(* Logix 5000 project; controller ARS14002_PLC vendor 1 type 14 code 218 rev 30.11; software revision 30.01; part 9 of 13 *)
(* tags used below, declared in another part *)
   AN_1000A : CM_AI_SCL;
   AN_1000A_RESTART_TMR : TIMER;
   AN_1000A_SP : REAL;
   AN_1000A_SPL : REAL;
   AN_1000A_STOP_TMR : TIMER;
   AN_1000B : CM_AI_SCL;
   AN_1000B_RESTART_TMR : TIMER;
   AN_1000B_SP : REAL;
   AN_1000B_SPL : REAL;
   AN_1000B_STOP_TMR : TIMER;
   ARS_DERIME_AUTO : BOOL;
   ARS_DERIME_AUTO_OSF_OB : BOOL;
   ARS_DERIME_AUTO_OSF_SB : BOOL;
   ARS_RETURN_AUTO : BOOL;
   AT2_ATOMIZE_FLOW_SCFM : REAL;
   AT2_INLET_FLOW_SCFM : REAL;
   AT2_NONATOMIZE_FLOW : REAL;
   AT2_PLANT_ATOMIZING : BOOL;
   AT2_PLANT_RETURN_AUTO : BOOL;
   AT3_ATOMIZE_FLOW_SCFM : REAL;
   AT3_INLET_FLOW_SCFM : REAL;
   AT3_NONATOMIZE_FLOW : REAL;
   AT3_PLANT_ATOMIZING : BOOL;
   AT3_PLANT_RETURN_AUTO : BOOL;
   BLENDING_OVERRIDE : BOOL;
   CALC_AN_1000B_BLENDED : REAL;
   CALC_HMI_FLOW : REAL;
   CP_Hi_Press_Shutoff : BOOL;
   DEOXO_ARGON_PURGE_DEPRESS : BOOL;
   DEOXO_ARGON_PURGE_FILL : BOOL;
   DEOXO_ARGON_PURGE_HIFLOW : BOOL;
   DEOXO_ARGON_PURGE_LOFLOW : BOOL;
   Deoxo_CurrentState : DINT;
   DEOXO_DEPRESS_TON : TIMER;
   DEOXO_DRY_REM : DINT;
   DEOXO_DRY_TON : TIMER;
   DEOXO_EXOTHERM_SP : REAL;
   DEOXO_OVERTEMP : BOOL;
   DEOXO_OVERTEMP_SPH : REAL;
   DEOXO_OVERTEMP_SPL : REAL;
   DEOXO_POST_EXO_REM : DINT;
   DEOXO_POST_EXOTHERM_TON : TIMER;
   DEOXO_PREHEAT_SP : REAL;
   DEOXO_PURGE_CYC_REM : DINT;
   DEOXO_PURGE_CYCLE_CTU : COUNTER;
   DEOXO_REGEN_HMI_BIT : BOOL;
   DEOXO_REGEN_HMI_BIT_ONS_F : BOOL;
   DEOXO_REGEN_HMI_BIT_ONS_R : BOOL;
   DEOXO_REGEN_RESET : BOOL;
   DEOXO_REGEN_RESET_ONS : BOOL;
   DEOXO_REGEN_RUN : BOOL;
   DEOXO_REGEN_START_PB : BOOL;
   DEOXO_REGEN_STOP_PB : BOOL;
   Deoxo_TransitionState : DINT;
   DEOXO_VENT_SPL : REAL;
   DEOXO_VENT_SWITCH_SP : REAL;
   EN_1250 : BOOL;   // HXR-1250 Enable Signal
   ESTOP_TRIP : BOOL;
   FCV_1001_ENABLE_TON : TIMER;
   FCV_1001_STARTPOS : REAL;
   FCV_1002_Atomize_Mode : BOOL;
   FCV_1002_FLOW_MODE : BOOL;   // 1 = FLOW CONTROL FT-1002 0 = PRESSURE CONTROL PT-1003
   FCV_1002_FLOW_MODE_AN_100B_PPM_MAX : REAL;
   FCV_1002_FLOW_MODE_MIN_FLOW : REAL;
   FCV_1002_FLOW_MODE_N2_PPM_SP : REAL;
   FCV_1002_FLOW_NOT_ATOMIZE_SP : REAL;
   FCV_1002_FLOW_SP : REAL;
   FCV_1002_FLOW_SP_AUTO : BOOL;
   FCV_1002_HIGHPRESS_MAXOPEN : REAL;
   FCV_1002_PT_1003_HIGHALM : BOOL;
   FCV_1002_PT_1003_HIGHLIM : REAL;
   FCV_1002_PT_1003_HIGHLIM_RESET : REAL;
   FCV_1002_PVSWITCH_AUTO : BOOL;
   FCV_1002_SP_Atomize : REAL;
   FCV_1002_SP_Idle_Standby : REAL;
   FCV_1002_STARTPOS : REAL;
   FT_1002 : CM_AI_SCL;
   FT_1002_MAVE : REAL;
   FT_202_ALT_SCFM : REAL;
   HXR_1250 : CM_DO_FVNR;
   LP_SHUTOFF_SPL : REAL;
   MODE_ATOMIZE : BOOL;
   P_800A_Start_Vent_TMR : TIMER;
   P_800B_Start_Vent_TMR : TIMER;
   PIDE_1001 : PID_ENHANCED;
   PIDE_1002 : PID_ENHANCED;
   PIDE_1002_FLOW_IGAIN : REAL;
   PIDE_1002_FLOW_PGAIN : REAL;
   PIDE_1002_FLOW_SP : PID_ENHANCED;
   PIDE_1002_PRESSURE_IGAIN : REAL;
   PIDE_1002_PRESSURE_PGAIN : REAL;
   PIDE_1002_PVCHANGE0 : BOOL;
   PIDE_1002_PVCHANGE1 : BOOL;
   PIDE_1002_RESET : BOOL;
   PIDE_1221 : PID_ENHANCED;
   PIDE_1251 : PID_ENHANCED;
   PIDE_800 : PID_ENHANCED;
   PIDE_800_InRange : BOOL;
   PILOT_PLANT_ATOMIZING : BOOL;
   PILOT_PLANT_RETURN_AUTO : BOOL;
   PRAX_N2_ASSUME : REAL;
   PT_1001 : CM_AI_SCL;
   PT_1001_MINUS_10 : REAL;
   PT_1001_MINUS_50 : REAL;
   PT_1003 : CM_AI_SCL;
   PT_1201 : CM_AI_SCL;
   PT_1301A : CM_AI_SCL;
   PT_902 : CM_AI_SCL;
   PWHMI_StartAtomizing : TIMER;
   Return_Stop_N2 : BOOL;
   Return_Stop_O2 : BOOL;
   SV_1001F : CM_DO_GENERIC;
   SV_1002F : CM_DO_GENERIC;
   SV_1207X : CM_DO_GENERIC;
   SV_1208X : CM_DO_GENERIC;
   SV_1221F : CM_DO_GENERIC;
   SV_1251F : CM_DO_GENERIC;
   TE_1201 : CM_AI_SCL;
   TE_1202 : CM_AI_SCL;
   TE_1203 : CM_AI_SCL;
   TE_901 : CM_AI_SCL;
   TE_901_InRange : BOOL;
   TE_901_SPH : REAL;
   TE_901_SPL : REAL;
   TE_902 : CM_AI_SCL;
   VFD_800A_EN : BOOL;
   VFD_800B_EN : BOOL;
   XV_1001 : CM_DO_VLV;
   XV_1201 : CM_DO_VLV;
   XV_1202 : CM_DO_VLV;
   XV_1203 : CM_DO_VLV;
   XV_1204 : CM_DO_VLV;
   XV_1205 : CM_DO_VLV;
(* MainProgram, continued *)

ROUTINE _306_HP_Product   (* ladder *)
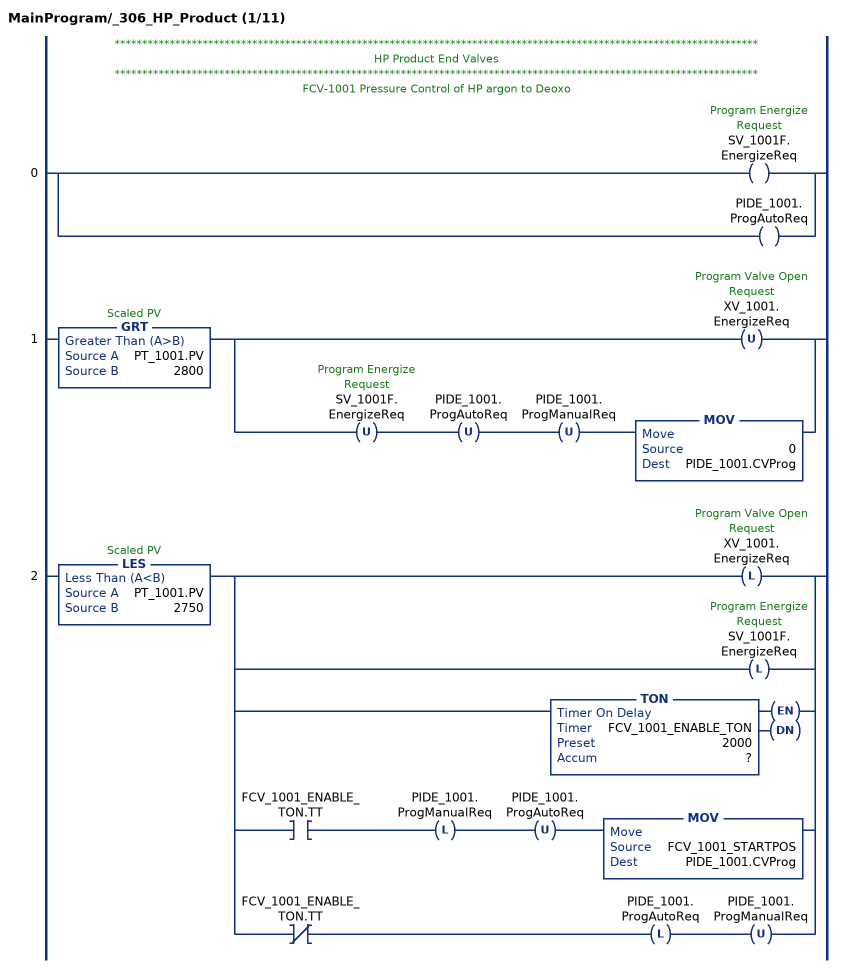
   // *********************************************************************************************************************
   // HP Product End Valves
   // *********************************************************************************************************************
   // FCV-1001 Pressure Control of HP argon to Deoxo
   0: [OTE(SV_1001F.EnergizeReq) ,OTE(PIDE_1001.ProgAutoReq) ];
   1: GRT(PT_1001.PV,2800)[OTU(XV_1001.EnergizeReq) ,OTU(SV_1001F.EnergizeReq) OTU(PIDE_1001.ProgAutoReq) OTU(PIDE_1001.ProgManualReq) MOV(0,PIDE_1001.CVProg) ];
   2: LES(PT_1001.PV,2750)[OTL(XV_1001.EnergizeReq) ,OTL(SV_1001F.EnergizeReq) ,TON(FCV_1001_ENABLE_TON,?,?) ,XIC(FCV_1001_ENABLE_TON.TT) OTL(PIDE_1001.ProgManualReq) OTU(PIDE_1001.ProgAutoReq) MOV(FCV_1001_STARTPOS,PIDE_1001.CVProg) ,XIO(FCV_1001_ENABLE_TON.TT) OTL(PIDE_1001.ProgAutoReq) OTU(PIDE_1001.ProgManualReq) ];
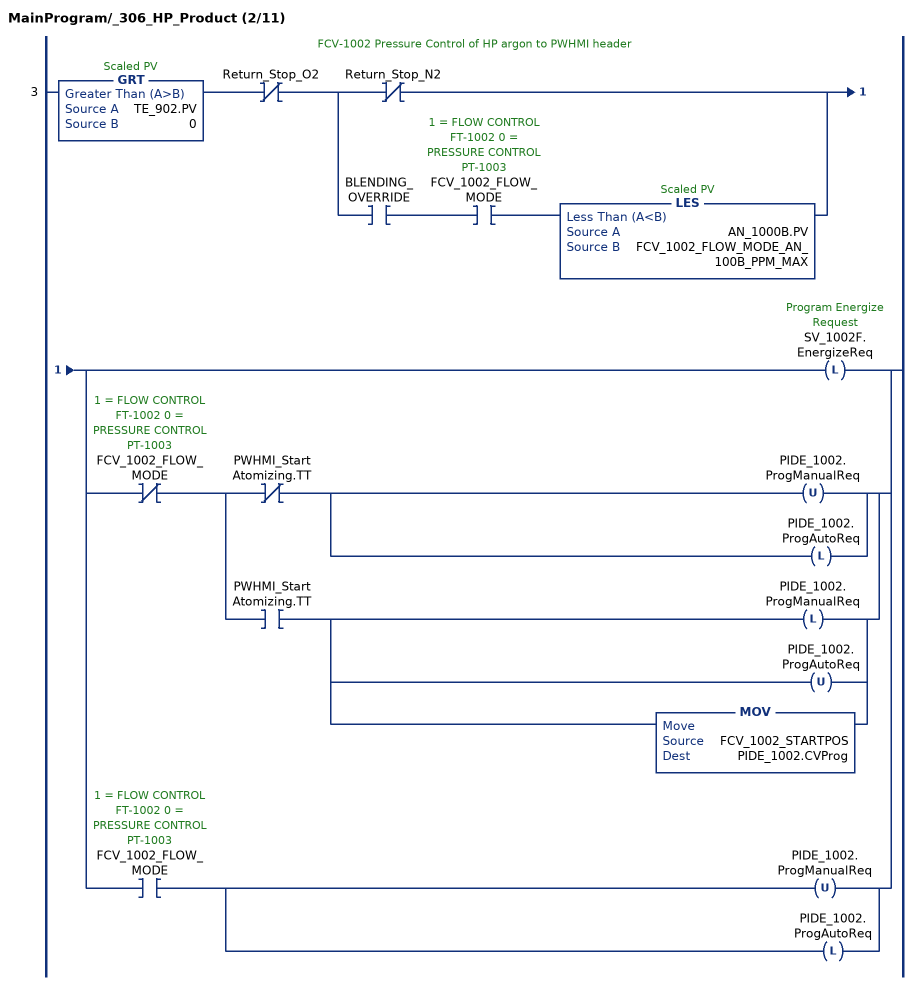
   // FCV-1002 Pressure Control of HP argon to PWHMI header
   3: GRT(TE_902.PV,0)XIO(Return_Stop_O2)[XIO(Return_Stop_N2) ,XIC(BLENDING_OVERRIDE) XIC(FCV_1002_FLOW_MODE) LES(AN_1000B.PV,FCV_1002_FLOW_MODE_AN_100B_PPM_MAX) ][OTL(SV_1002F.EnergizeReq) ,XIO(FCV_1002_FLOW_MODE) [XIO(PWHMI_StartAtomizing.TT) [OTU(PIDE_1002.ProgManualReq) ,OTL(PIDE_1002.ProgAutoReq) ] ,XIC(PWHMI_StartAtomizing.TT) [OTL(PIDE_1002.ProgManualReq) ,OTU(PIDE_1002.ProgAutoReq) ,MOV(FCV_1002_STARTPOS,PIDE_1002.CVProg) ] ] ,XIC(FCV_1002_FLOW_MODE) [OTU(PIDE_1002.ProgManualReq) ,OTL(PIDE_1002.ProgAutoReq) ] ];
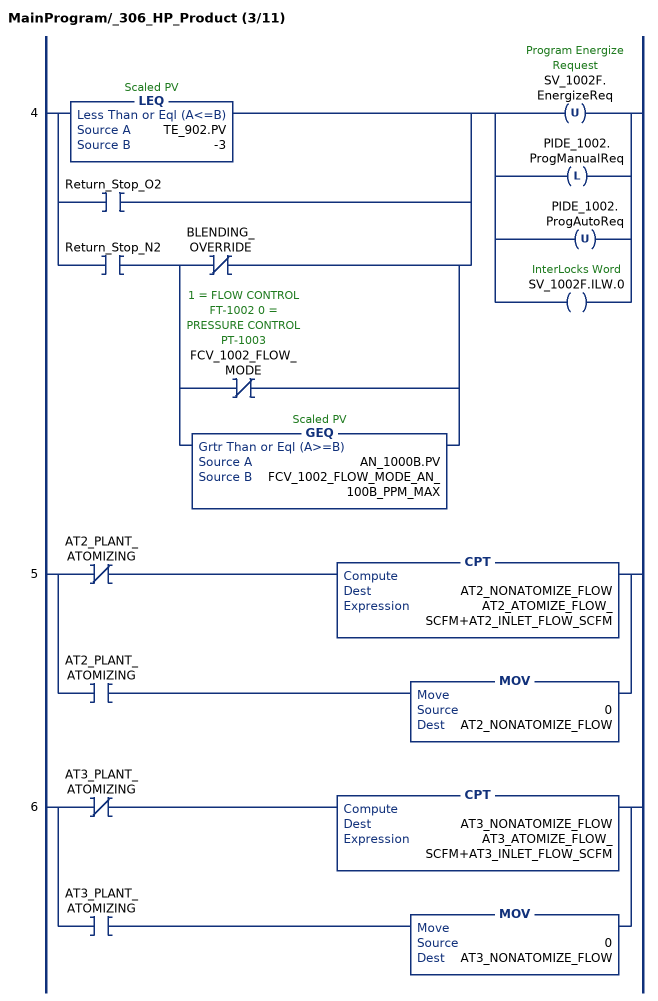
   4: [LEQ(TE_902.PV,-3) ,XIC(Return_Stop_O2) ,XIC(Return_Stop_N2) [XIO(BLENDING_OVERRIDE) ,XIO(FCV_1002_FLOW_MODE) ,GEQ(AN_1000B.PV,FCV_1002_FLOW_MODE_AN_100B_PPM_MAX) ] ][OTU(SV_1002F.EnergizeReq) ,OTL(PIDE_1002.ProgManualReq) ,OTU(PIDE_1002.ProgAutoReq) ,OTE(SV_1002F.ILW.0) ];
   5: [XIO(AT2_PLANT_ATOMIZING) CPT(AT2_NONATOMIZE_FLOW,AT2_ATOMIZE_FLOW_SCFM+AT2_INLET_FLOW_SCFM) ,XIC(AT2_PLANT_ATOMIZING) MOV(0,AT2_NONATOMIZE_FLOW) ];
   6: [XIO(AT3_PLANT_ATOMIZING) CPT(AT3_NONATOMIZE_FLOW,AT3_ATOMIZE_FLOW_SCFM+AT3_INLET_FLOW_SCFM) ,XIC(AT3_PLANT_ATOMIZING) MOV(0,AT3_NONATOMIZE_FLOW) ];
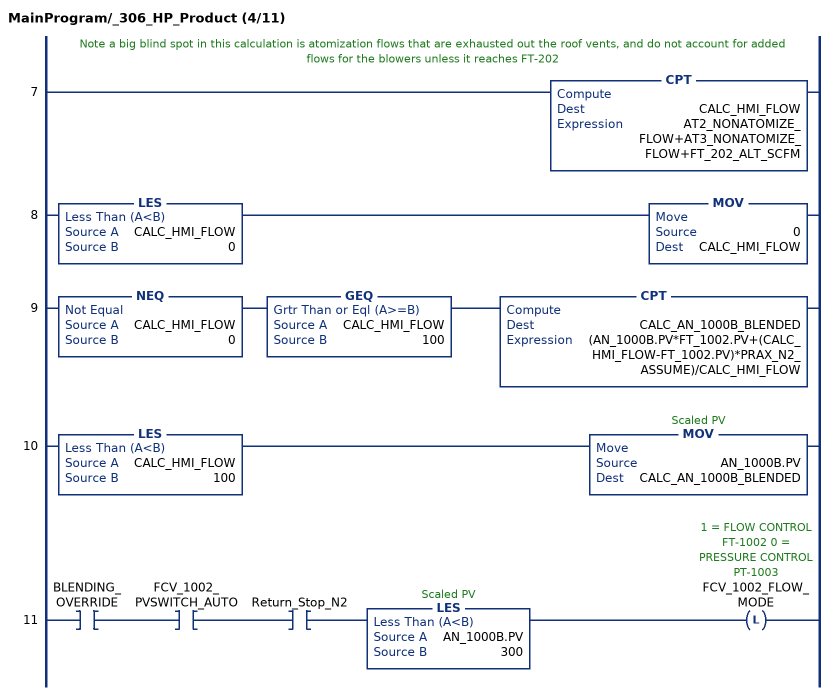
   // Note a big blind spot in this calculation is atomization flows that are exhausted out the roof vents, and do not account for added flows for the blowers unless it reaches FT-202
   7: CPT(CALC_HMI_FLOW,AT2_NONATOMIZE_FLOW+AT3_NONATOMIZE_FLOW+FT_202_ALT_SCFM);
   8: LES(CALC_HMI_FLOW,0)MOV(0,CALC_HMI_FLOW);
   9: NEQ(CALC_HMI_FLOW,0)GEQ(CALC_HMI_FLOW,100)CPT(CALC_AN_1000B_BLENDED,(AN_1000B.PV*FT_1002.PV+(CALC_HMI_FLOW-FT_1002.PV)*PRAX_N2_ASSUME)/CALC_HMI_FLOW);
   10: LES(CALC_HMI_FLOW,100)MOV(AN_1000B.PV,CALC_AN_1000B_BLENDED);
   11: XIC(BLENDING_OVERRIDE)XIC(FCV_1002_PVSWITCH_AUTO)XIC(Return_Stop_N2)LES(AN_1000B.PV,300)OTL(FCV_1002_FLOW_MODE);
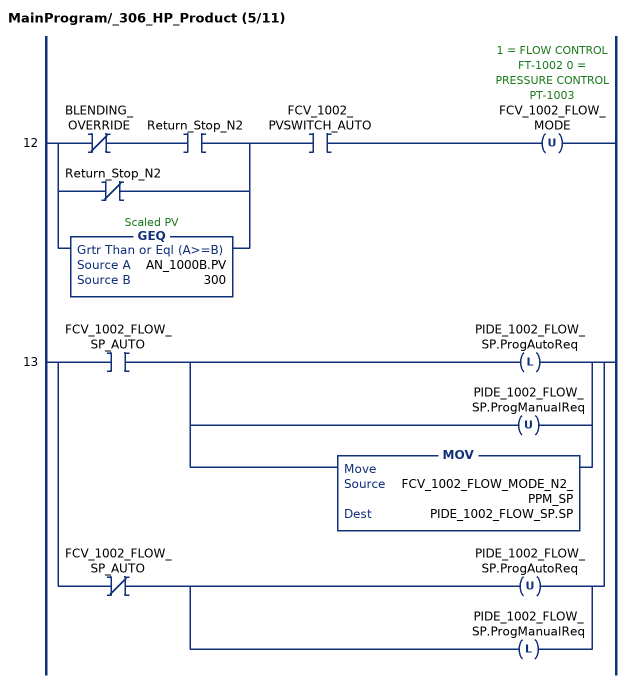
   12: [XIO(BLENDING_OVERRIDE) XIC(Return_Stop_N2) ,XIO(Return_Stop_N2) ,GEQ(AN_1000B.PV,300) ]XIC(FCV_1002_PVSWITCH_AUTO)OTU(FCV_1002_FLOW_MODE);
   13: [XIC(FCV_1002_FLOW_SP_AUTO) [OTL(PIDE_1002_FLOW_SP.ProgAutoReq) ,OTU(PIDE_1002_FLOW_SP.ProgManualReq) ,MOV(FCV_1002_FLOW_MODE_N2_PPM_SP,PIDE_1002_FLOW_SP.SP) ] ,XIO(FCV_1002_FLOW_SP_AUTO) [OTU(PIDE_1002_FLOW_SP.ProgAutoReq) ,OTL(PIDE_1002_FLOW_SP.ProgManualReq) ] ];
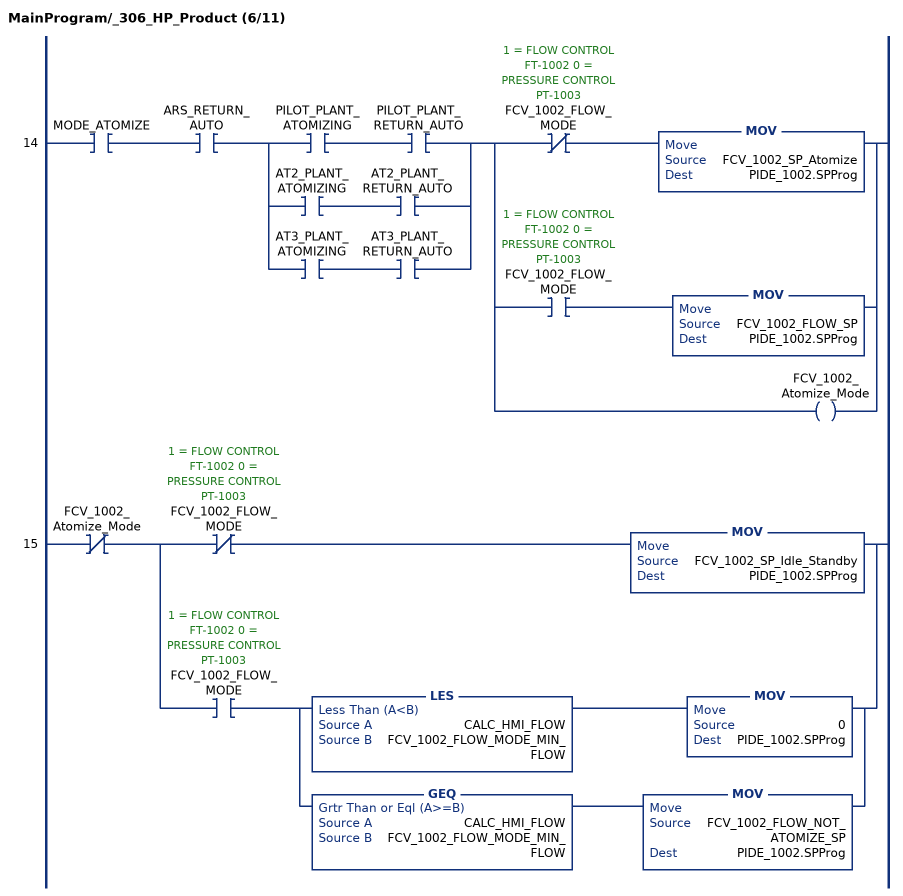
   14: XIC(MODE_ATOMIZE)XIC(ARS_RETURN_AUTO)[XIC(PILOT_PLANT_ATOMIZING) XIC(PILOT_PLANT_RETURN_AUTO) ,XIC(AT2_PLANT_ATOMIZING) XIC(AT2_PLANT_RETURN_AUTO) ,XIC(AT3_PLANT_ATOMIZING) XIC(AT3_PLANT_RETURN_AUTO) ][XIO(FCV_1002_FLOW_MODE) MOV(FCV_1002_SP_Atomize,PIDE_1002.SPProg) ,XIC(FCV_1002_FLOW_MODE) MOV(FCV_1002_FLOW_SP,PIDE_1002.SPProg) ,OTE(FCV_1002_Atomize_Mode) ];
   15: XIO(FCV_1002_Atomize_Mode)[XIO(FCV_1002_FLOW_MODE) MOV(FCV_1002_SP_Idle_Standby,PIDE_1002.SPProg) ,XIC(FCV_1002_FLOW_MODE) [LES(CALC_HMI_FLOW,FCV_1002_FLOW_MODE_MIN_FLOW) MOV(0,PIDE_1002.SPProg) ,GEQ(CALC_HMI_FLOW,FCV_1002_FLOW_MODE_MIN_FLOW) MOV(FCV_1002_FLOW_NOT_ATOMIZE_SP,PIDE_1002.SPProg) ] ];
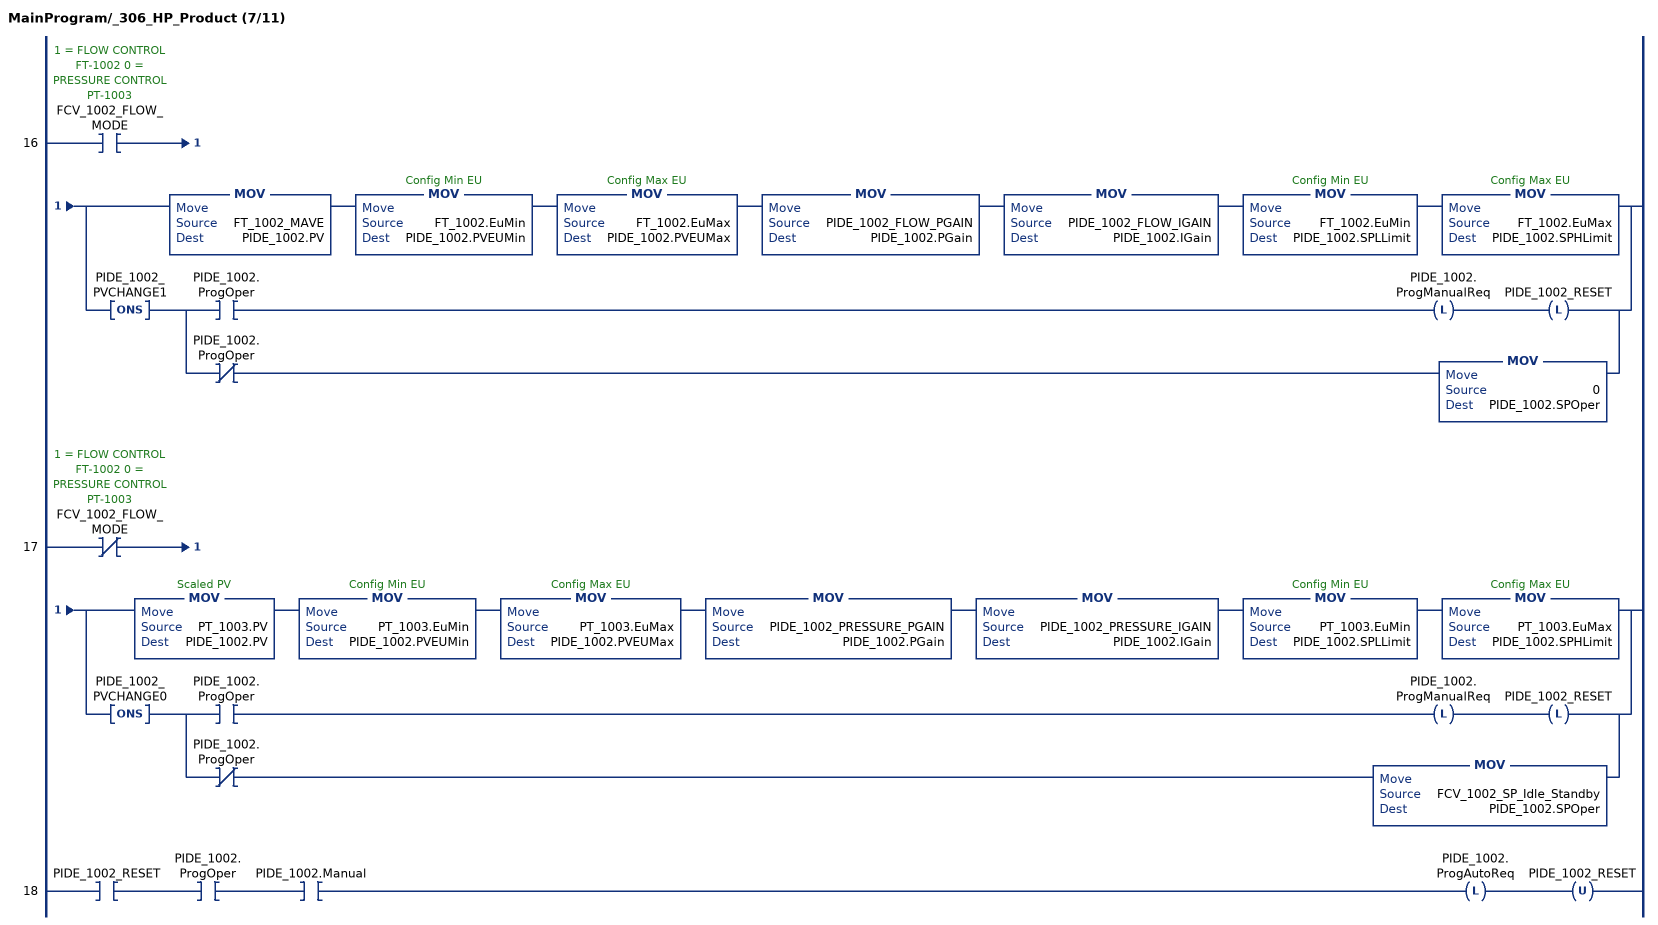
   16: XIC(FCV_1002_FLOW_MODE)[MOV(FT_1002_MAVE,PIDE_1002.PV) MOV(FT_1002.EuMin,PIDE_1002.PVEUMin) MOV(FT_1002.EuMax,PIDE_1002.PVEUMax) MOV(PIDE_1002_FLOW_PGAIN,PIDE_1002.PGain) MOV(PIDE_1002_FLOW_IGAIN,PIDE_1002.IGain) MOV(FT_1002.EuMin,PIDE_1002.SPLLimit) MOV(FT_1002.EuMax,PIDE_1002.SPHLimit) ,ONS(PIDE_1002_PVCHANGE1) [XIC(PIDE_1002.ProgOper) OTL(PIDE_1002.ProgManualReq) OTL(PIDE_1002_RESET) ,XIO(PIDE_1002.ProgOper) MOV(0,PIDE_1002.SPOper) ] ];
   17: XIO(FCV_1002_FLOW_MODE)[MOV(PT_1003.PV,PIDE_1002.PV) MOV(PT_1003.EuMin,PIDE_1002.PVEUMin) MOV(PT_1003.EuMax,PIDE_1002.PVEUMax) MOV(PIDE_1002_PRESSURE_PGAIN,PIDE_1002.PGain) MOV(PIDE_1002_PRESSURE_IGAIN,PIDE_1002.IGain) MOV(PT_1003.EuMin,PIDE_1002.SPLLimit) MOV(PT_1003.EuMax,PIDE_1002.SPHLimit) ,ONS(PIDE_1002_PVCHANGE0) [XIC(PIDE_1002.ProgOper) OTL(PIDE_1002.ProgManualReq) OTL(PIDE_1002_RESET) ,XIO(PIDE_1002.ProgOper) MOV(FCV_1002_SP_Idle_Standby,PIDE_1002.SPOper) ] ];
   18: XIC(PIDE_1002_RESET)XIC(PIDE_1002.ProgOper)XIC(PIDE_1002.Manual)OTL(PIDE_1002.ProgAutoReq)OTU(PIDE_1002_RESET);
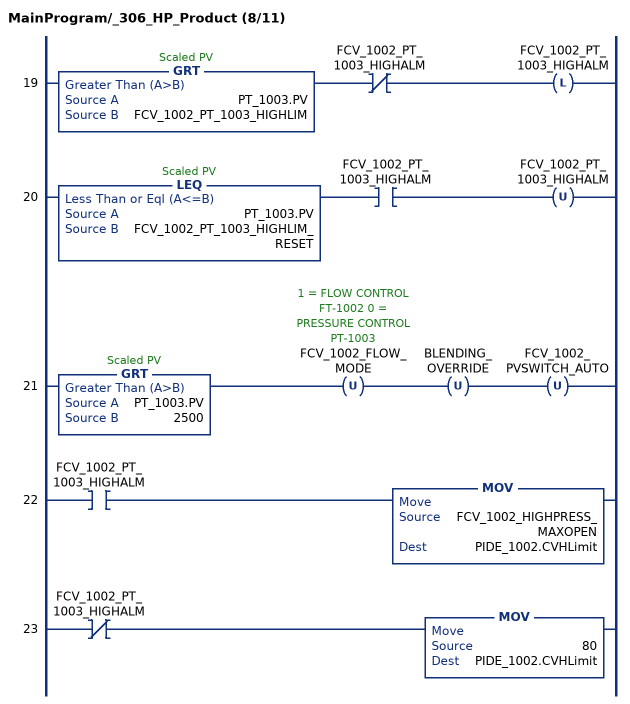
   19: GRT(PT_1003.PV,FCV_1002_PT_1003_HIGHLIM)XIO(FCV_1002_PT_1003_HIGHALM)OTL(FCV_1002_PT_1003_HIGHALM);
   20: LEQ(PT_1003.PV,FCV_1002_PT_1003_HIGHLIM_RESET)XIC(FCV_1002_PT_1003_HIGHALM)OTU(FCV_1002_PT_1003_HIGHALM);
   21: GRT(PT_1003.PV,2500)OTU(FCV_1002_FLOW_MODE)OTU(BLENDING_OVERRIDE)OTU(FCV_1002_PVSWITCH_AUTO);
   22: XIC(FCV_1002_PT_1003_HIGHALM)MOV(FCV_1002_HIGHPRESS_MAXOPEN,PIDE_1002.CVHLimit);
   23: XIO(FCV_1002_PT_1003_HIGHALM)MOV(80,PIDE_1002.CVHLimit);
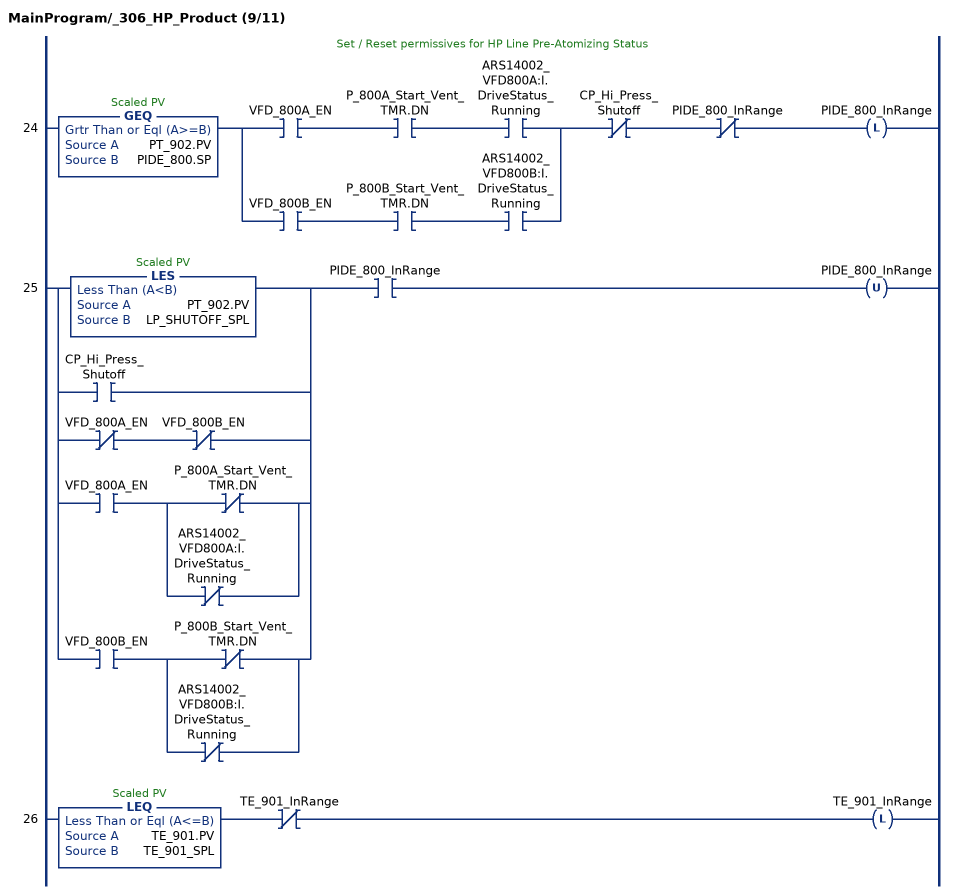
   // Set / Reset permissives for HP Line Pre-Atomizing Status
   24: GEQ(PT_902.PV,PIDE_800.SP)[XIC(VFD_800A_EN) XIC(P_800A_Start_Vent_TMR.DN) XIC(ARS14002_VFD800A:I.DriveStatus_Running) ,XIC(VFD_800B_EN) XIC(P_800B_Start_Vent_TMR.DN) XIC(ARS14002_VFD800B:I.DriveStatus_Running) ]XIO(CP_Hi_Press_Shutoff)XIO(PIDE_800_InRange)OTL(PIDE_800_InRange);
   25: [LES(PT_902.PV,LP_SHUTOFF_SPL) ,XIC(CP_Hi_Press_Shutoff) ,XIO(VFD_800A_EN) XIO(VFD_800B_EN) ,XIC(VFD_800A_EN) [XIO(P_800A_Start_Vent_TMR.DN) ,XIO(ARS14002_VFD800A:I.DriveStatus_Running) ] ,XIC(VFD_800B_EN) [XIO(P_800B_Start_Vent_TMR.DN) ,XIO(ARS14002_VFD800B:I.DriveStatus_Running) ] ]XIC(PIDE_800_InRange)OTU(PIDE_800_InRange);
   26: LEQ(TE_901.PV,TE_901_SPL)XIO(TE_901_InRange)OTL(TE_901_InRange);
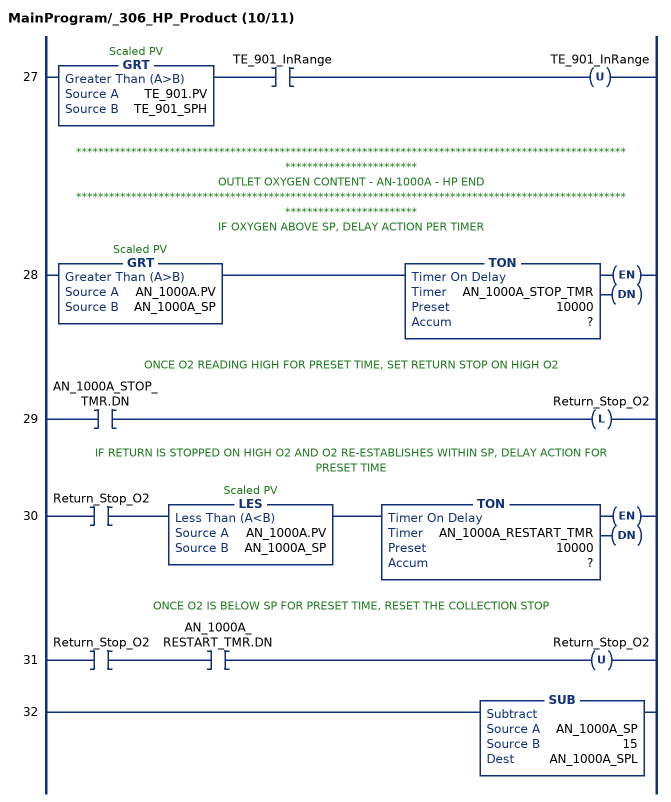
   27: GRT(TE_901.PV,TE_901_SPH)XIC(TE_901_InRange)OTU(TE_901_InRange);
   // ****************************************************************************************************************************
   // OUTLET OXYGEN CONTENT - AN-1000A - HP END
   // ****************************************************************************************************************************
   // IF OXYGEN ABOVE SP, DELAY ACTION PER TIMER
   28: GRT(AN_1000A.PV,AN_1000A_SP)TON(AN_1000A_STOP_TMR,?,?);
   // ONCE O2 READING HIGH FOR PRESET TIME, SET RETURN STOP ON HIGH O2
   29: XIC(AN_1000A_STOP_TMR.DN)OTL(Return_Stop_O2);
   // IF RETURN IS STOPPED ON HIGH O2 AND O2 RE-ESTABLISHES WITHIN SP, DELAY ACTION FOR PRESET TIME
   30: XIC(Return_Stop_O2)LES(AN_1000A.PV,AN_1000A_SP)TON(AN_1000A_RESTART_TMR,?,?);
   // ONCE O2 IS BELOW SP FOR PRESET TIME, RESET THE COLLECTION STOP
   31: XIC(Return_Stop_O2)XIC(AN_1000A_RESTART_TMR.DN)OTU(Return_Stop_O2);
   32: SUB(AN_1000A_SP,15,AN_1000A_SPL);
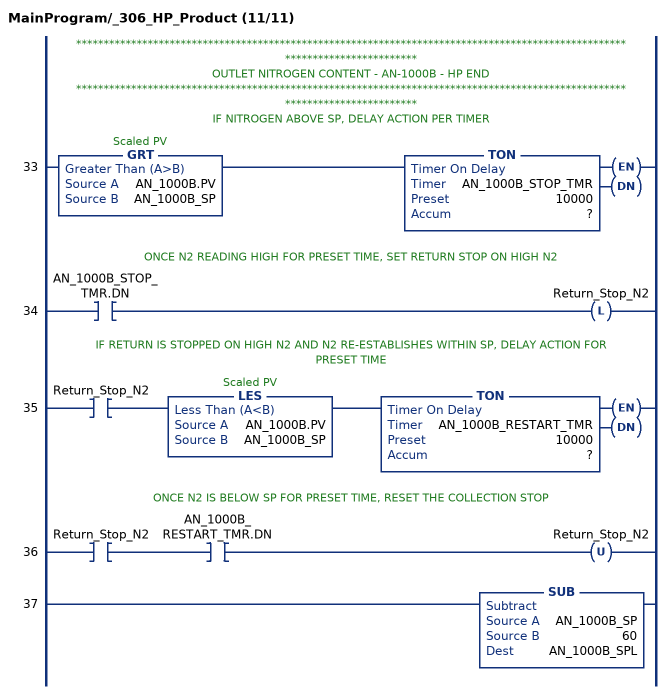
   // ****************************************************************************************************************************
   // OUTLET NITROGEN CONTENT - AN-1000B - HP END
   // ****************************************************************************************************************************
   // IF NITROGEN ABOVE SP, DELAY ACTION PER TIMER
   33: GRT(AN_1000B.PV,AN_1000B_SP)TON(AN_1000B_STOP_TMR,?,?);
   // ONCE N2 READING HIGH FOR PRESET TIME, SET RETURN STOP ON HIGH N2
   34: XIC(AN_1000B_STOP_TMR.DN)OTL(Return_Stop_N2);
   // IF RETURN IS STOPPED ON HIGH N2 AND N2 RE-ESTABLISHES WITHIN SP, DELAY ACTION FOR PRESET TIME
   35: XIC(Return_Stop_N2)LES(AN_1000B.PV,AN_1000B_SP)TON(AN_1000B_RESTART_TMR,?,?);
   // ONCE N2 IS BELOW SP FOR PRESET TIME, RESET THE COLLECTION STOP
   36: XIC(Return_Stop_N2)XIC(AN_1000B_RESTART_TMR.DN)OTU(Return_Stop_N2);
   37: SUB(AN_1000B_SP,60,AN_1000B_SPL);
END_ROUTINE

ROUTINE _307_Deoxo   (* ladder *)
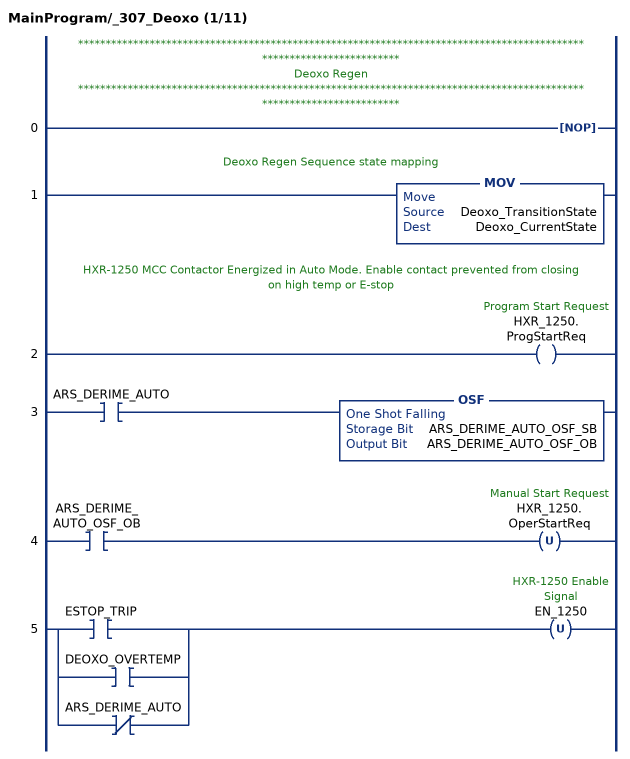
   // *********************************************************************************************************************
   // Deoxo Regen
   // *********************************************************************************************************************
   0: NOP();
   // Deoxo Regen Sequence state mapping
   1: MOV(Deoxo_TransitionState,Deoxo_CurrentState);
   // HXR-1250 MCC Contactor Energized in Auto Mode. Enable contact prevented from closing on high temp or E-stop
   2: OTE(HXR_1250.ProgStartReq);
   3: XIC(ARS_DERIME_AUTO)OSF(ARS_DERIME_AUTO_OSF_SB,ARS_DERIME_AUTO_OSF_OB);
   4: XIC(ARS_DERIME_AUTO_OSF_OB)OTU(HXR_1250.OperStartReq);
   5: [XIC(ESTOP_TRIP) ,XIC(DEOXO_OVERTEMP) ,XIO(ARS_DERIME_AUTO) ]OTU(EN_1250);
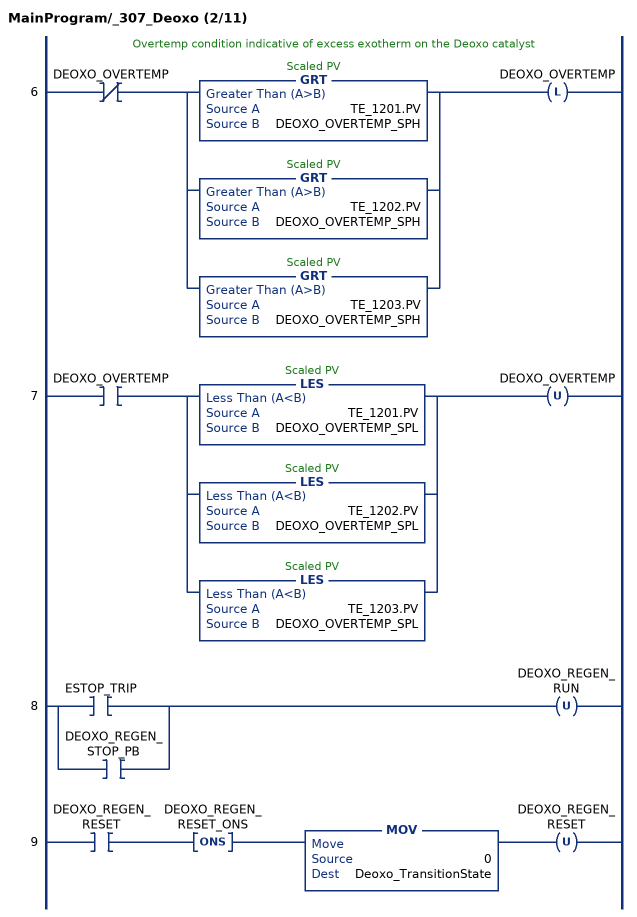
   // Overtemp condition indicative of excess exotherm on the Deoxo catalyst
   6: XIO(DEOXO_OVERTEMP)[GRT(TE_1201.PV,DEOXO_OVERTEMP_SPH) ,GRT(TE_1202.PV,DEOXO_OVERTEMP_SPH) ,GRT(TE_1203.PV,DEOXO_OVERTEMP_SPH) ]OTL(DEOXO_OVERTEMP);
   7: XIC(DEOXO_OVERTEMP)[LES(TE_1201.PV,DEOXO_OVERTEMP_SPL) ,LES(TE_1202.PV,DEOXO_OVERTEMP_SPL) ,LES(TE_1203.PV,DEOXO_OVERTEMP_SPL) ]OTU(DEOXO_OVERTEMP);
   8: [XIC(ESTOP_TRIP) ,XIC(DEOXO_REGEN_STOP_PB) ]OTU(DEOXO_REGEN_RUN);
   9: XIC(DEOXO_REGEN_RESET)ONS(DEOXO_REGEN_RESET_ONS)MOV(0,Deoxo_TransitionState)OTU(DEOXO_REGEN_RESET);
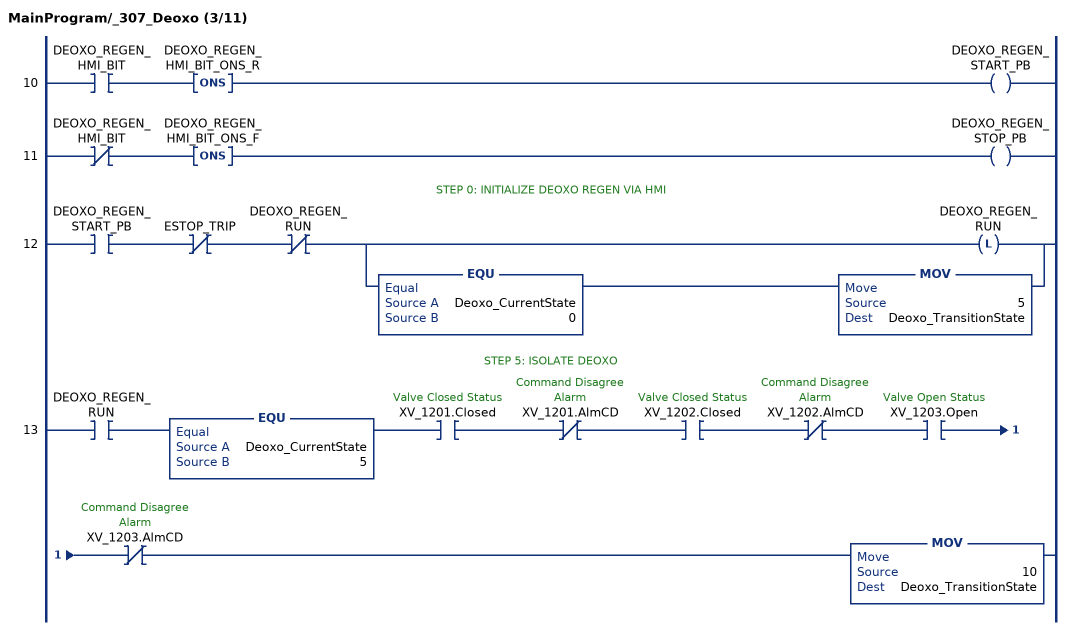
   10: XIC(DEOXO_REGEN_HMI_BIT)ONS(DEOXO_REGEN_HMI_BIT_ONS_R)OTE(DEOXO_REGEN_START_PB);
   11: XIO(DEOXO_REGEN_HMI_BIT)ONS(DEOXO_REGEN_HMI_BIT_ONS_F)OTE(DEOXO_REGEN_STOP_PB);
   // STEP 0: INITIALIZE DEOXO REGEN VIA HMI
   12: XIC(DEOXO_REGEN_START_PB)XIO(ESTOP_TRIP)XIO(DEOXO_REGEN_RUN)[OTL(DEOXO_REGEN_RUN) ,EQU(Deoxo_CurrentState,0) MOV(5,Deoxo_TransitionState) ];
   // STEP 5: ISOLATE DEOXO
   13: XIC(DEOXO_REGEN_RUN)EQU(Deoxo_CurrentState,5)XIC(XV_1201.Closed)XIO(XV_1201.AlmCD)XIC(XV_1202.Closed)XIO(XV_1202.AlmCD)XIC(XV_1203.Open)XIO(XV_1203.AlmCD)MOV(10,Deoxo_TransitionState);
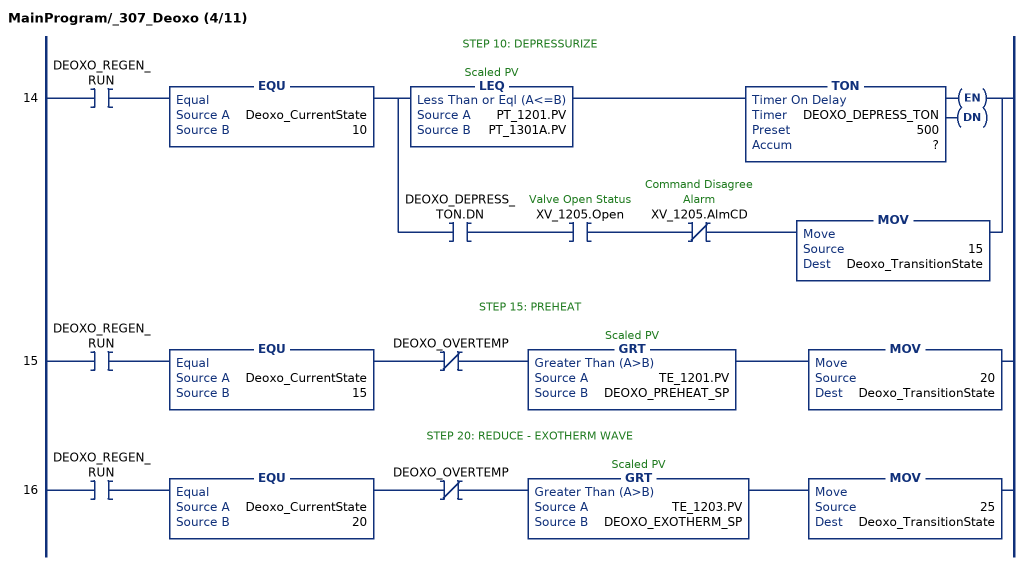
   // STEP 10: DEPRESSURIZE
   14: XIC(DEOXO_REGEN_RUN)EQU(Deoxo_CurrentState,10)[LEQ(PT_1201.PV,PT_1301A.PV) TON(DEOXO_DEPRESS_TON,?,?) ,XIC(DEOXO_DEPRESS_TON.DN) XIC(XV_1205.Open) XIO(XV_1205.AlmCD) MOV(15,Deoxo_TransitionState) ];
   // STEP 15: PREHEAT
   15: XIC(DEOXO_REGEN_RUN)EQU(Deoxo_CurrentState,15)XIO(DEOXO_OVERTEMP)GRT(TE_1201.PV,DEOXO_PREHEAT_SP)MOV(20,Deoxo_TransitionState);
   // STEP 20: REDUCE - EXOTHERM WAVE
   16: XIC(DEOXO_REGEN_RUN)EQU(Deoxo_CurrentState,20)XIO(DEOXO_OVERTEMP)GRT(TE_1203.PV,DEOXO_EXOTHERM_SP)MOV(25,Deoxo_TransitionState);
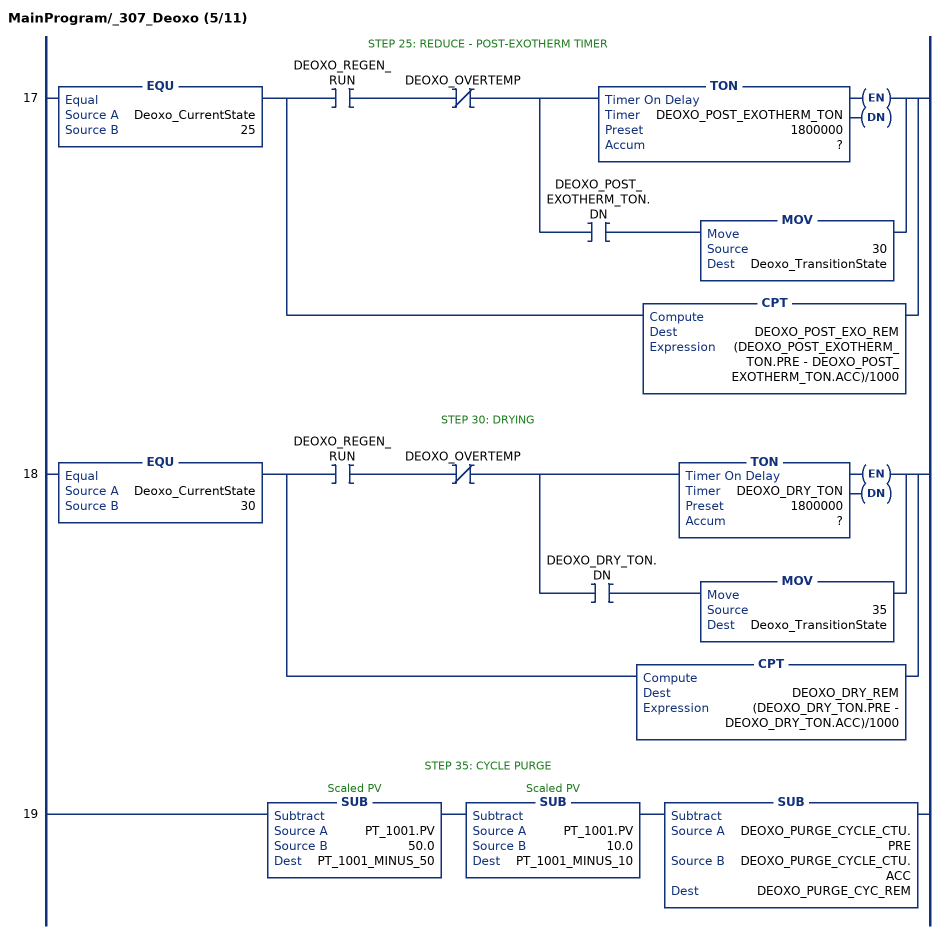
   // STEP 25: REDUCE - POST-EXOTHERM TIMER
   17: EQU(Deoxo_CurrentState,25)[XIC(DEOXO_REGEN_RUN) XIO(DEOXO_OVERTEMP) [TON(DEOXO_POST_EXOTHERM_TON,?,?) ,XIC(DEOXO_POST_EXOTHERM_TON.DN) MOV(30,Deoxo_TransitionState) ] ,CPT(DEOXO_POST_EXO_REM,(DEOXO_POST_EXOTHERM_TON.PRE - DEOXO_POST_EXOTHERM_TON.ACC)/1000) ];
   // STEP 30: DRYING
   18: EQU(Deoxo_CurrentState,30)[XIC(DEOXO_REGEN_RUN) XIO(DEOXO_OVERTEMP) [TON(DEOXO_DRY_TON,?,?) ,XIC(DEOXO_DRY_TON.DN) MOV(35,Deoxo_TransitionState) ] ,CPT(DEOXO_DRY_REM,(DEOXO_DRY_TON.PRE - DEOXO_DRY_TON.ACC)/1000) ];
   // STEP 35: CYCLE PURGE
   19: SUB(PT_1001.PV,50.0,PT_1001_MINUS_50)SUB(PT_1001.PV,10.0,PT_1001_MINUS_10)SUB(DEOXO_PURGE_CYCLE_CTU.PRE,DEOXO_PURGE_CYCLE_CTU.ACC,DEOXO_PURGE_CYC_REM);
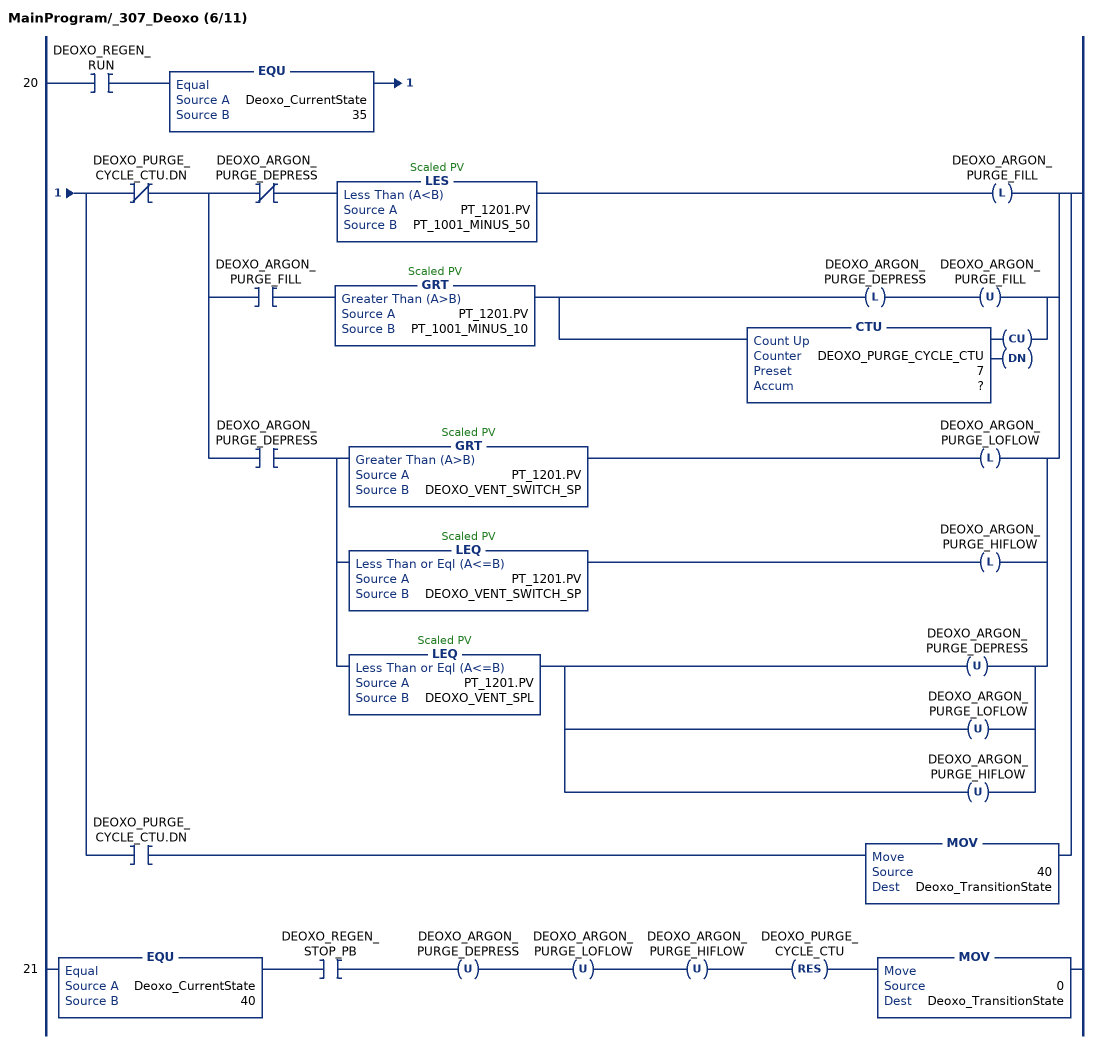
   20: XIC(DEOXO_REGEN_RUN)EQU(Deoxo_CurrentState,35)[XIO(DEOXO_PURGE_CYCLE_CTU.DN) [XIO(DEOXO_ARGON_PURGE_DEPRESS) LES(PT_1201.PV,PT_1001_MINUS_50) OTL(DEOXO_ARGON_PURGE_FILL) ,XIC(DEOXO_ARGON_PURGE_FILL) GRT(PT_1201.PV,PT_1001_MINUS_10) [OTL(DEOXO_ARGON_PURGE_DEPRESS) OTU(DEOXO_ARGON_PURGE_FILL) ,CTU(DEOXO_PURGE_CYCLE_CTU,?,?) ] ,XIC(DEOXO_ARGON_PURGE_DEPRESS) [GRT(PT_1201.PV,DEOXO_VENT_SWITCH_SP) OTL(DEOXO_ARGON_PURGE_LOFLOW) ,LEQ(PT_1201.PV,DEOXO_VENT_SWITCH_SP) OTL(DEOXO_ARGON_PURGE_HIFLOW) ,LEQ(PT_1201.PV,DEOXO_VENT_SPL) [OTU(DEOXO_ARGON_PURGE_DEPRESS) ,OTU(DEOXO_ARGON_PURGE_LOFLOW) ,OTU(DEOXO_ARGON_PURGE_HIFLOW) ] ] ] ,XIC(DEOXO_PURGE_CYCLE_CTU.DN) MOV(40,Deoxo_TransitionState) ];
   21: EQU(Deoxo_CurrentState,40)XIC(DEOXO_REGEN_STOP_PB)OTU(DEOXO_ARGON_PURGE_DEPRESS)OTU(DEOXO_ARGON_PURGE_LOFLOW)OTU(DEOXO_ARGON_PURGE_HIFLOW)RES(DEOXO_PURGE_CYCLE_CTU)MOV(0,Deoxo_TransitionState);
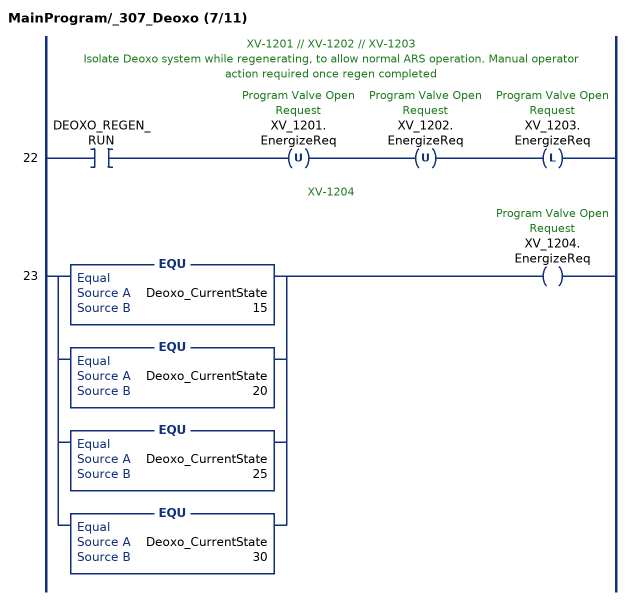
   // XV-1201 // XV-1202 // XV-1203
   // Isolate Deoxo system while regenerating, to allow normal ARS operation. Manual operator action required once regen completed
   22: XIC(DEOXO_REGEN_RUN)OTU(XV_1201.EnergizeReq)OTU(XV_1202.EnergizeReq)OTL(XV_1203.EnergizeReq);
   // XV-1204
   23: [EQU(Deoxo_CurrentState,15) ,EQU(Deoxo_CurrentState,20) ,EQU(Deoxo_CurrentState,25) ,EQU(Deoxo_CurrentState,30) ]OTE(XV_1204.EnergizeReq);
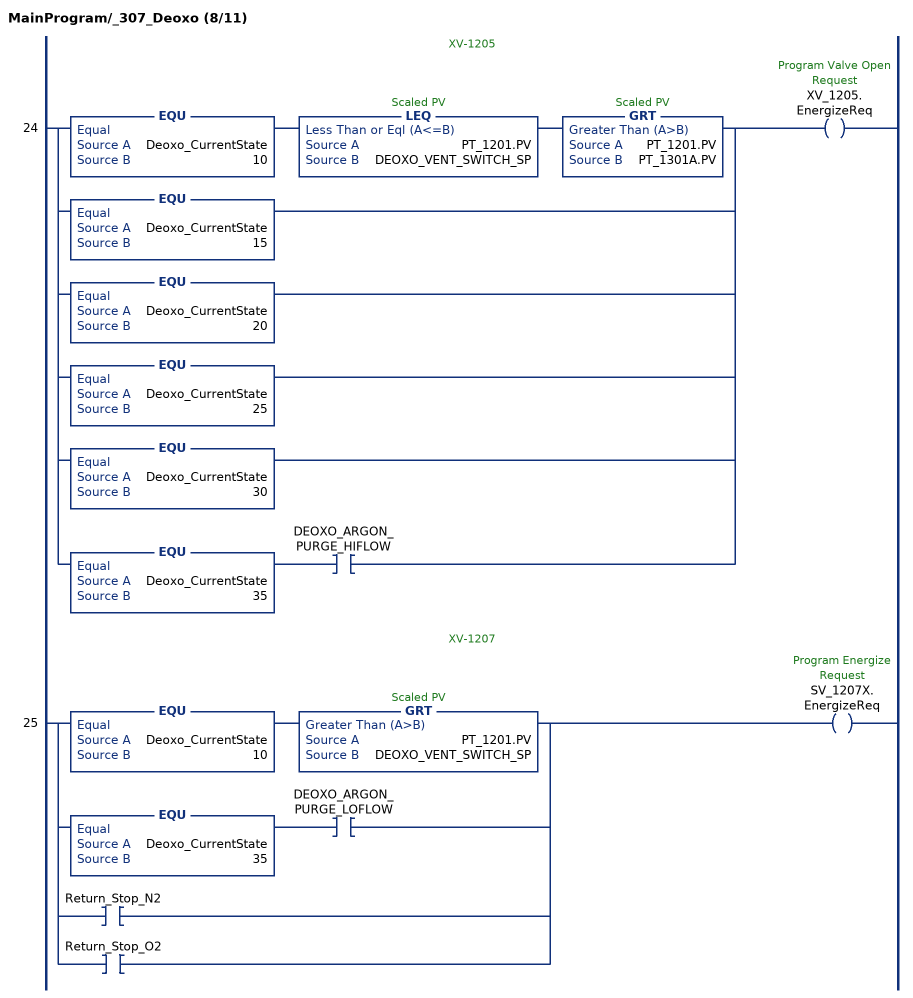
   // XV-1205
   24: [EQU(Deoxo_CurrentState,10) LEQ(PT_1201.PV,DEOXO_VENT_SWITCH_SP) GRT(PT_1201.PV,PT_1301A.PV) ,EQU(Deoxo_CurrentState,15) ,EQU(Deoxo_CurrentState,20) ,EQU(Deoxo_CurrentState,25) ,EQU(Deoxo_CurrentState,30) ,EQU(Deoxo_CurrentState,35) XIC(DEOXO_ARGON_PURGE_HIFLOW) ]OTE(XV_1205.EnergizeReq);
   // XV-1207
   25: [EQU(Deoxo_CurrentState,10) GRT(PT_1201.PV,DEOXO_VENT_SWITCH_SP) ,EQU(Deoxo_CurrentState,35) XIC(DEOXO_ARGON_PURGE_LOFLOW) ,XIC(Return_Stop_N2) ,XIC(Return_Stop_O2) ]OTE(SV_1207X.EnergizeReq);
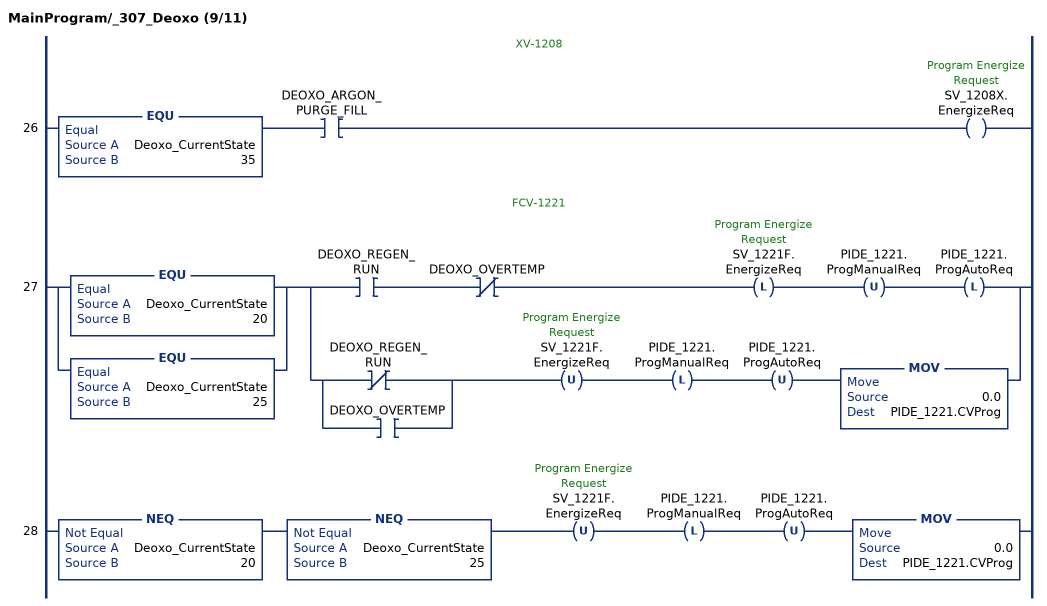
   // XV-1208
   26: EQU(Deoxo_CurrentState,35)XIC(DEOXO_ARGON_PURGE_FILL)OTE(SV_1208X.EnergizeReq);
   // FCV-1221
   27: [EQU(Deoxo_CurrentState,20) ,EQU(Deoxo_CurrentState,25) ][XIC(DEOXO_REGEN_RUN) XIO(DEOXO_OVERTEMP) OTL(SV_1221F.EnergizeReq) OTU(PIDE_1221.ProgManualReq) OTL(PIDE_1221.ProgAutoReq) ,[XIO(DEOXO_REGEN_RUN) ,XIC(DEOXO_OVERTEMP) ] OTU(SV_1221F.EnergizeReq) OTL(PIDE_1221.ProgManualReq) OTU(PIDE_1221.ProgAutoReq) MOV(0.0,PIDE_1221.CVProg) ];
   28: NEQ(Deoxo_CurrentState,20)NEQ(Deoxo_CurrentState,25)OTU(SV_1221F.EnergizeReq)OTL(PIDE_1221.ProgManualReq)OTU(PIDE_1221.ProgAutoReq)MOV(0.0,PIDE_1221.CVProg);
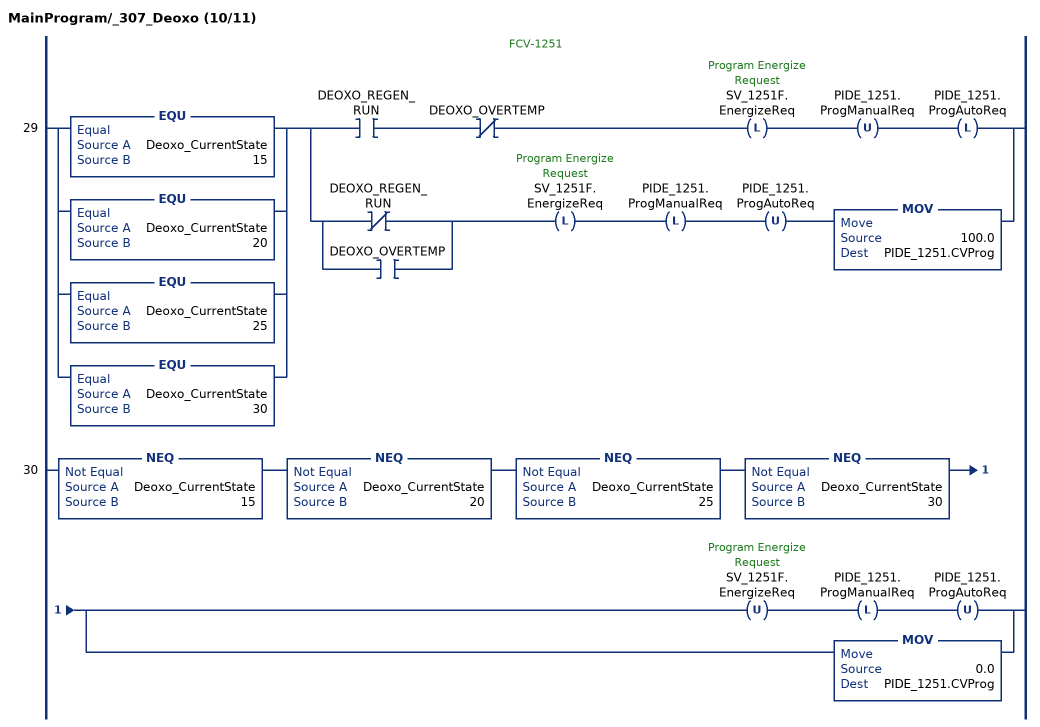
   // FCV-1251
   29: [EQU(Deoxo_CurrentState,15) ,EQU(Deoxo_CurrentState,20) ,EQU(Deoxo_CurrentState,25) ,EQU(Deoxo_CurrentState,30) ][XIC(DEOXO_REGEN_RUN) XIO(DEOXO_OVERTEMP) OTL(SV_1251F.EnergizeReq) OTU(PIDE_1251.ProgManualReq) OTL(PIDE_1251.ProgAutoReq) ,[XIO(DEOXO_REGEN_RUN) ,XIC(DEOXO_OVERTEMP) ] OTL(SV_1251F.EnergizeReq) OTL(PIDE_1251.ProgManualReq) OTU(PIDE_1251.ProgAutoReq) MOV(100.0,PIDE_1251.CVProg) ];
   30: NEQ(Deoxo_CurrentState,15)NEQ(Deoxo_CurrentState,20)NEQ(Deoxo_CurrentState,25)NEQ(Deoxo_CurrentState,30)[OTU(SV_1251F.EnergizeReq) OTL(PIDE_1251.ProgManualReq) OTU(PIDE_1251.ProgAutoReq) ,MOV(0.0,PIDE_1251.CVProg) ];
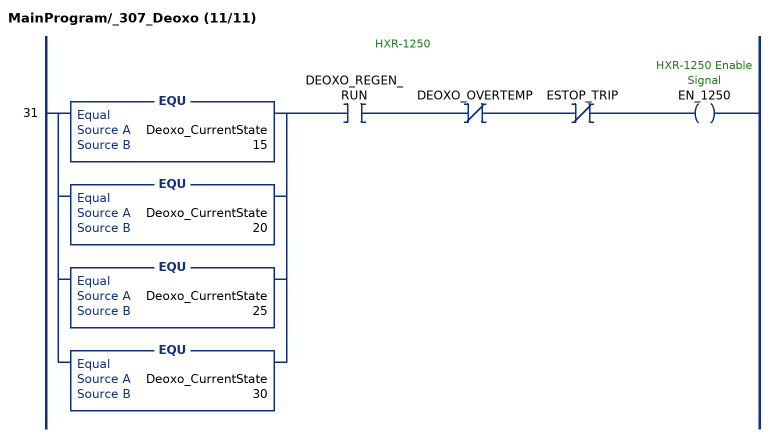
   // HXR-1250
   31: [EQU(Deoxo_CurrentState,15) ,EQU(Deoxo_CurrentState,20) ,EQU(Deoxo_CurrentState,25) ,EQU(Deoxo_CurrentState,30) ]XIC(DEOXO_REGEN_RUN)XIO(DEOXO_OVERTEMP)XIO(ESTOP_TRIP)OTE(EN_1250);
END_ROUTINE
